// TIA Portal V18 export
// export: Created 2026-06-03T15:33:17.742158Z, ExportSetting WithDefaults
Screen "06_Chung_Cat_Tu_Dong"  800x600, Number=6
  ScreenLayer "Layer_0"
    GraphicView "SCADA_Background_Graphic" at 0,0 size 800x600  Picture=scada_distillation_bg
    GraphicIOField "GFX_V101" at 330,455 size 44x38  Mode=Output, OnValue=1, PictureList=GL_Van_Hoi
      ProcessValue := HMI_SteamValve_GFX
    Button "Btn_V101_Transparent" at 330,455 size 44x38  Mode=Text
      on Click: InvertBit(Tag := Van_Cap_Hoi_M)
    GraphicIOField "GFX_V102" at 520,125 size 48x29  Mode=Output, OnValue=1, PictureList=GL_Van_Xa
      ProcessValue := HMI_DrainValve_GFX
    IOField "IO_Feed_Level" at 225,310 size 55x22  DataFormat=Decimal, FormatPattern=99.9, Mode=Output
      ProcessValue := Muc_Nuoc_PV
    IOField "IO_Col_Temp" at 500,485 size 55x22  DataFormat=Decimal, FormatPattern=999.9, Mode=Output
      ProcessValue := Nhiet_Do_PV
    GraphicIOField "GFX_Alarm" at 10,10 size 54x43  Mode=Output, OnValue=1, PictureList=GL_Alarm
      ProcessValue := HMI_Alarm_GFX
    Button "Nav_Btn_1" at 27,529 size 107x46  Mode=Text, TextOff="TỔNG QUAN"
      on Click: ActivateScreen(Screen name := 01_Tong_Quan, Object number := 0)
    Button "Nav_Btn_2" at 147,529 size 107x46  Mode=Text, TextOff="VẬN HÀNH"
      on Click: ActivateScreen(Screen name := 02_Van_Hanh, Object number := 0)
    Button "Nav_Btn_3" at 267,529 size 107x46  Mode=Text, TextOff="PID & NƯỚC"
      on Click: ActivateScreen(Screen name := 03_PID_Muc_Nuoc, Object number := 0)
    Button "Nav_Btn_4" at 387,529 size 107x46  Mode=Text, TextOff="TREND"
      on Click: ActivateScreen(Screen name := 04_Trend, Object number := 0)
    Button "Nav_Btn_5" at 507,529 size 107x46  Mode=Text, TextOff="CẢNH BÁO"
      on Click: ActivateScreen(Screen name := 05_Canh_Bao_IO, Object number := 0)
    Button "Nav_Btn_6" at 627,529 size 107x46  Mode=Text, TextOff="CHƯNG CẤT"
    Button "Nav_Exit_Btn" at 732,552 size 65x30  Mode=Text, TextOff="EXIT"
      on Click: StopRuntime(Mode := 0)
